FUNCTION_BLOCK MoveModuloMoverToPosition EXTENDS TaskBase
VAR_INPUT
END_VAR
VAR_OUTPUT
END_VAR
VAR
	moveAbs	: MC_MoveAbsoluteCA;
	_axis : REFERENCE TO AXIS_REF;
	_MoveMover : BOOL;
	_stOptions : ST_MoveAbsoluteCAOptions;
END_VAR

METHOD Abort : BOOL
moveAbs.Execute := FALSE;
moveAbs.Position := moveAbs.Velocity := 0;
_MoveMover := false;
_busy := false;
Abort := true;
State := 0;
END_METHOD

PROPERTY PUBLIC Acceleration : mc_lreal
GET
Acceleration := moveAbs.Acceleration;
END_GET
SET
moveAbs.Acceleration := Acceleration;
END_SET
END_PROPERTY

METHOD Cycle : BOOL
VAR_INPUT
END_VAR
CASE State OF
	0:
		IF _MoveMover THEN
			_done := FALSE;
			_error := FALSE;
			_busy := TRUE;
			moveAbs.Execute := TRUE;
			IF moveAbs.Busy THEN
				State := 10;
				_MoveMover := FALSE;
			END_IF
		END_IF
		
	10:
		IF NOT moveAbs.Busy THEN
			IF moveAbs.Done THEN
				_done := TRUE;
			ELSIF moveAbs.Error THEN
				_error := TRUE;
			END_IF
			_busy := FALSE;
			moveAbs.Execute := FALSE;
			State := 0;
		END_IF
END_CASE

moveAbs(Axis := _axis, Options := _stOptions);
END_METHOD

PROPERTY PUBLIC Deceleration : mc_lreal
GET
Deceleration := moveAbs.Deceleration;
END_GET
SET
moveAbs.Deceleration := Deceleration;
END_SET
END_PROPERTY

METHOD FB_init : BOOL
VAR_INPUT
	bInitRetains : BOOL; // if TRUE, the retain variables are initialized (warm start / cold start)
	bInCopyCode : BOOL;  // if TRUE, the instance afterwards gets moved into the copy code (online change)
	axis : reference TO AXIS_REF;
END_VAR
_axis REF= axis;
END_METHOD

PROPERTY PUBLIC Gap : mc_lreal
GET
Gap := moveAbs.Gap;
END_GET
SET
moveAbs.Gap := Gap;
END_SET
END_PROPERTY

PROPERTY PUBLIC Jerk : mc_lreal
GET
Jerk := moveAbs.Jerk;
END_GET
SET
moveAbs.Jerk := Jerk;
END_SET
END_PROPERTY

METHOD MoveTo : BOOL
VAR_INPUT
	Position : MC_LREAL;
	Velocity : MC_LREAL;
	Direction: Tc3_Mc3Definitions.MC_DIRECTION;
	Turns: UDINT;
END_VAR
moveAbs.Position := Position;
moveAbs.Velocity := Velocity;
moveAbs.Direction := Direction;
moveAbs.Options.AdditionalTurns := Turns;
_MoveMover := MoveTo := true;
END_METHOD

PROPERTY PUBLIC Options : ST_MoveAbsoluteCAOptions
GET
Options := _stOptions;
END_GET
SET
_stOptions := Options;
END_SET
END_PROPERTY

END_FUNCTION_BLOCK

(* stored: Version 1.1.0.1, ProductVersion 3.1.4024.12
   POU MoveModuloMoverToPosition: Id {86a89fc0-d952-4342-8bc4-3e7afaf8d6b0}, SpecialFunc None
   Method Abort: Id {5c5502fe-cfbb-4721-939d-6b8391fd3812}
   Property Acceleration: Id {bd8e2346-8872-4feb-ac95-f472cf2ca2c7}
   Get Get: Id {c4ef743d-06c1-4445-9890-b82ffba396f1}
   Set Set: Id {1c8827c9-2f8f-4b77-8024-4b0046d69ac2}
   Method Cycle: Id {4cb00213-de2b-40d2-a495-86e25cb3d039}
   Property Deceleration: Id {9b084d4a-e02d-4702-912a-4bc5910ddae2}
   Get Get: Id {a47d2d08-c000-41b9-a1f9-a582ebe1b9d1}
   Set Set: Id {82a7f264-1036-48b4-a621-2fa4d8fd0895}
   Method FB_init: Id {37fbed4c-5b49-4a9c-886b-a9cda5653c34}
   Property Gap: Id {6f40f3be-1ac5-4f41-a512-900c33b72e2e}
   Get Get: Id {d520ecb2-c250-4598-84bd-dc6b0a2aef6c}
   Set Set: Id {49d06445-a9cb-4b50-a172-a728c79a3bc7}
   Property Jerk: Id {557e6884-85fe-4a0b-9fbe-e021e4eb6165}
   Get Get: Id {43424688-9bf6-468e-9d81-7307bd08e1b7}
   Set Set: Id {fbdecc92-c967-41e0-99c8-b2c9f3bf8bd0}
   Method MoveTo: Id {42a523a0-ad8a-4fac-a76b-d1875ec2f808}
   Property Options: Id {1dd7fc51-dd5a-4f57-a3ca-696f6637a39e}
   Get Get: Id {179a8440-f33d-4396-9725-56d6b0191700}
   Set Set: Id {18307288-77cd-4621-a1f2-e62bd90c9ccf} *)
